FUNCTION_BLOCK FB_TapVariable
////////////////// 
// TAp a variable when input is active and reset after 
//////////////////	

VAR_IN_OUT
	TapOut			: BOOL;		// Output VTap Variable
	
END_VAR

VAR_INPUT
	TapTrigger		: BOOL;		// Input Trigger
	
END_VAR

VAR
	F_TRIG_Trigger	: F_TRIG;	// Trigger detection 
	R_TRIG_Trigger	: R_TRIG;	// Trigger detection 		
	
	
END_VAR

R_TRIG_Trigger(CLK:= TapTrigger);
F_TRIG_Trigger(CLK:= TapTrigger);

IF R_TRIG_Trigger.Q THEN
	TapOut			:=TRUE;
	
ELSIF F_TRIG_Trigger.Q  THEN 
	TapOut			:=FALSE ;
			
END_IF

END_FUNCTION_BLOCK

(* stored: Version 1.1.0.1, ProductVersion 3.1.4024.6
   POU FB_TapVariable: Id {25ee244e-7237-4fd7-acd2-d23945c1121c}, SpecialFunc None *)
